// TIA Portal V18 export
DATA_BLOCK "HOOTER_DB_1"   // DB102
VERSION : 0.1
// stored: AutoNumber true, DBAccessibleFromOPCUA true, DBAccessibleFromWebserver true, InstanceOfName HOOTER, InstanceOfType FB
"HOOTER"
   // VAR_INPUT
   //    COND1 : Bool;
   //    COND2 : Bool;
   //    COND3 : Bool;
   //    COND4 : Bool;
   //    COND5 : Bool;
   //    COND6 : Bool;
   //    COND7 : Bool;
   //    COND8 : Bool;
   //    COND9 : Bool;
   //    COND10 : Bool;
   //    HOOTER_DI : Bool;
   // END_VAR
   // VAR_OUTPUT
   //    HOOTER_HMI : Bool;
   //    HOOTER_DO : Bool;
   // END_VAR
   // VAR_IN_OUT
   //    ACK : Bool;
   // END_VAR
   // VAR
   //    RS1 : Bool;
   //    RS2 : Bool;
   //    RS3 : Bool;
   //    RS4 : Bool;
   //    RS5 : Bool;
   //    RS6 : Bool;
   //    RS7 : Bool;
   //    RS8 : Bool;
   //    RS9 : Bool;
   //    RS10 : Bool;
   // END_VAR
BEGIN
END_DATA_BLOCK
